# EPICS alarm handler configuration: alh_files/mgnt_li25_kick.alhConfig
GROUP NULL KICK:LI25:MG01
   $COMMAND edm -x -eolc -noedit mgnt_li25_lgps.edl
$ALIAS KICK
$GUIDANCE
Li25 KICK Magnets
   Group Name: KICK:LI25:MG01
   Summary PV:  KICK:LI25:MG01:STATSUMY
$END

GROUP KICK:LI25:MG01  KICK:LI25:344
   $COMMAND edm -x -eolc -noedit -m "DEV=KICK:LI25:344" mgnt_unit.edl
CHANNEL   KICK:LI25:344       KICK:LI25:344:STATMSG                 -----
   $FORCEPV KICK:LI25:344:STATMSGSV -DATL 1 0
